FUNCTION Init_PB_Mom_125x100 : INT

VAR_INPUT
END_VAR

VAR

END_VAR

VAR_IN_OUT
	COMP:TS_Component;
END_VAR

COMP.B_TYPE:=0;
COMP.size:=0;

END_FUNCTION

(* stored: Version 1.1.0.1, ProductVersion 3.1.4020.12
   POU Init_PB_Mom_125x100: Id {b180adfe-f9bf-4340-a80f-5daa7bbf25c5}, SpecialFunc None *)
